FUNCTION_BLOCK AUDI2_I_TO_UDINT (* Composite FB for convert AUDI2 to UDINT *)
  (* Standard: 61499-2; Description: Copyright (c) 2024 HR Agrartechnik GmbH This program and the accompanying materials are made available under the terms of the Eclipse Public License 2.0 which is available at https://www.eclipse.org/legal/epl-2.0/ SPDX-License-Identifier: EPL-2.0 *)
  (* Version 1.0, 2026-09-12, Franz Höpfinger, HR Agrartechnik GmbH, Initial Version - Konvertierungsfamilie vervollstaendigt (analog zu AR2/AB2/AE2). *)
  PACKAGE adapter::conversion::bidirectional;
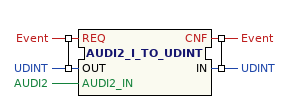
  EVENT_INPUT
    REQ WITH OUT; (* Request to Adapter *)
  END_EVENT
  EVENT_OUTPUT
    CNF WITH IN; (* Confirmation from Adapter *)
  END_EVENT
  VAR_INPUT
    OUT : UDINT;
  END_VAR
  VAR_OUTPUT
    IN : UDINT; (* Input data from Adapter *)
  END_VAR
  SOCKETS
    AUDI2_IN : adapter::types::bidirectional::AUDI2; (* Adapter Input *)
  END_SOCKETS
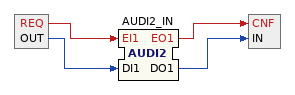
  EVENT_CONNECTIONS
    AUDI2_IN.EO1 TO CNF;
    REQ TO AUDI2_IN.EI1;
  END_CONNECTIONS
  DATA_CONNECTIONS
    AUDI2_IN.DO1 TO IN;
    OUT TO AUDI2_IN.DI1;
  END_CONNECTIONS
END_FUNCTION_BLOCK
